FUNCTION_BLOCK "G023G_Code"
TITLE =G023G GENERAL ELEMENTS KILN MALT TRANSFER
//COPYRIGHT:    (C) 2009  BUHLER AG, CH-9240 UZWIL, SWITZERLAND
//
//PRODUCT:      WinCoS_BIW01_09
//
//TITLE:        GENERAL ELEMENTS KILN MALT TRANSFER
//                General group control
//                Allgemeine Gruppensteuerung
//
//--------------------------------------------------------------------------------
//
//IDENT:        AUTHOR:             DEPT:                              DATE:
//
//P01_FB123.1.0 K.Renz              CSB41                              29.Sep.2009
//             1st Release
//
//--------------------------------------------------------------------------------
//
//PURPOSE:
//
//MANUAL :
//
//RESTRICTIONS:
//
//--------------------------------------------------------------------------------
AUTHOR : KR
FAMILY : USW
VERSION : 9.9


VAR
  Gr : "GCS7_GrpCtrlSub";	//Standard interface to group
  InOutValue1 : DINT ;	//Data for user
  InOutValue2 : DINT ;	//Data for user
  OutWayConflict : BOOL ;	//Data for user
  OutSelectionOk : BOOL ;	//Data for user
  CmdNewValue : BOOL ;	//Data for user
  CmdNewJob : BOOL ;	//Data for user
  OutCodeOK : BOOL ;	//Data for user
  InEndOfJob : BOOL ;	//Data for user
  staWayOk : BOOL ;	//Data for user
  EdgeStartRelease : BOOL ;	//Data for user
  USW8 : BOOL ;	//Data for user
  USW9 : BOOL ;	//Data for user
  USW10 : BOOL ;	//Data for user
  USW11 : BOOL ;	//Data for user
  USW12 : BOOL ;	//Data for user
  USW13 : BOOL ;	//Data for user
  USW14 : BOOL ;	//Data for user
  USW15 : BOOL ;	//Data for user
  A_3999_SHE01 : "GCS7_E_DigInput";	// DigInpCont
  A_3999_SHE02 : "GCS7_E_DigInput";	// DigInpCont
  A_39_A040Z1 : "GCS7_E_DigInput";	// DigInpCont
  A_39_A097Z1 : "GCS7_E_DigInput";	// DigInpCont
  A_39_A187Z1 : "GCS7_E_DigInput";	// DigInpCont
  A_39_A227Z1 : "GCS7_E_DigInput";	// DigInpCont
  A_39_K091Z1 : "GCS7_E_DigInput";	// DigInpCont
  A_39_S_H097 : "GCS7_E_DigInput";	// DigInpCont
END_VAR
VAR_TEMP
  tmpEnable : BOOL ;
  tmpFlag : BOOL ;
  tmpCmdNext : BOOL ;
  tmpLocal : BOOL ;
  tmpAspOk : BOOL ;
  tmpHWStop : BOOL ;
  tmpInstanzDBNo : INT ;
END_VAR
BEGIN
NETWORK
TITLE =



NETWORK
TITLE =Read command from group control
//Parameter
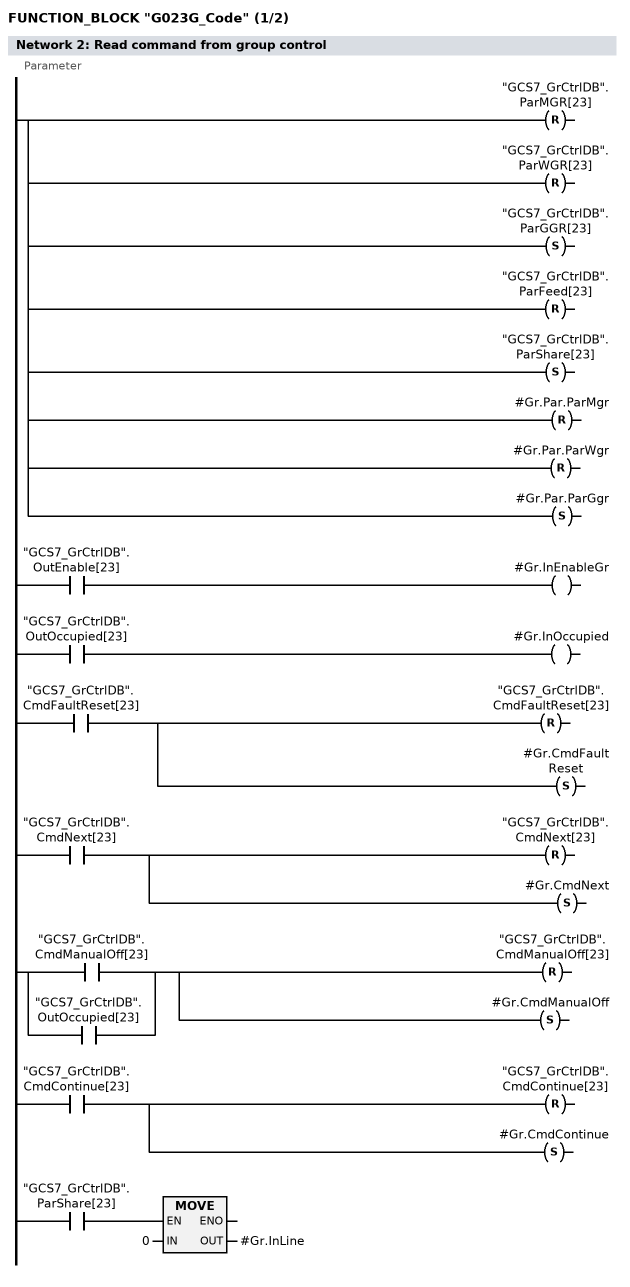
      SET   ;
      R     "GCS7_GrCtrlDB".ParMGR[23];
      R     "GCS7_GrCtrlDB".ParWGR[23];
      S     "GCS7_GrCtrlDB".ParGGR[23];
      R     "GCS7_GrCtrlDB".ParFeed[23];
      S     "GCS7_GrCtrlDB".ParShare[23];
      R     #Gr.Par.ParMgr;
      R     #Gr.Par.ParWgr;
      S     #Gr.Par.ParGgr;
//Command
      U     "GCS7_GrCtrlDB".OutEnable[23];
      =     #Gr.InEnableGr;
      U     "GCS7_GrCtrlDB".OutOccupied[23];
      =     #Gr.InOccupied;
      U     "GCS7_GrCtrlDB".CmdFaultReset[23];
      R     "GCS7_GrCtrlDB".CmdFaultReset[23];
      S     #Gr.CmdFaultReset;
      U     "GCS7_GrCtrlDB".CmdNext[23];
      R     "GCS7_GrCtrlDB".CmdNext[23];
      S     #Gr.CmdNext;
      U     "GCS7_GrCtrlDB".CmdManualOff[23];
      O     "GCS7_GrCtrlDB".OutOccupied[23];
      R     "GCS7_GrCtrlDB".CmdManualOff[23];
      S     #Gr.CmdManualOff;
      U     "GCS7_GrCtrlDB".CmdContinue[23];
      R     "GCS7_GrCtrlDB".CmdContinue[23];
      S     #Gr.CmdContinue;
//Init Line Number
      U     "GCS7_GrCtrlDB".ParShare[23];
      SPBN  WE00;
      L     0;
      T     #Gr.InLine;
WE00: NOP   0;
NETWORK
TITLE =Call Methode Control
// 1. Handle Interface PCControl
// 2. Prepare mode --> ModePassive,ModeActive,ModeIdling
// 3. Reset global flags of the group
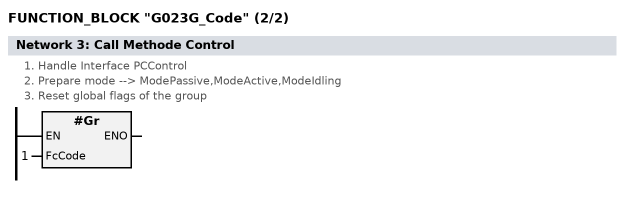
      CALL #Gr (
           FcCode                   := 1);
NETWORK
TITLE =Restart Idling Time

      CLR   ;
      S     #Gr.CmdRestartIdling;
NETWORK
TITLE =Prepare global flags



NETWORK
TITLE =Set Pattern (Target position)



NETWORK
TITLE =Interlocking WayOk



NETWORK
TITLE =Interlocking Autostart

      CLR   ;
      R     #Gr.OutAutostart;
NETWORK
TITLE =Interlocking Enable
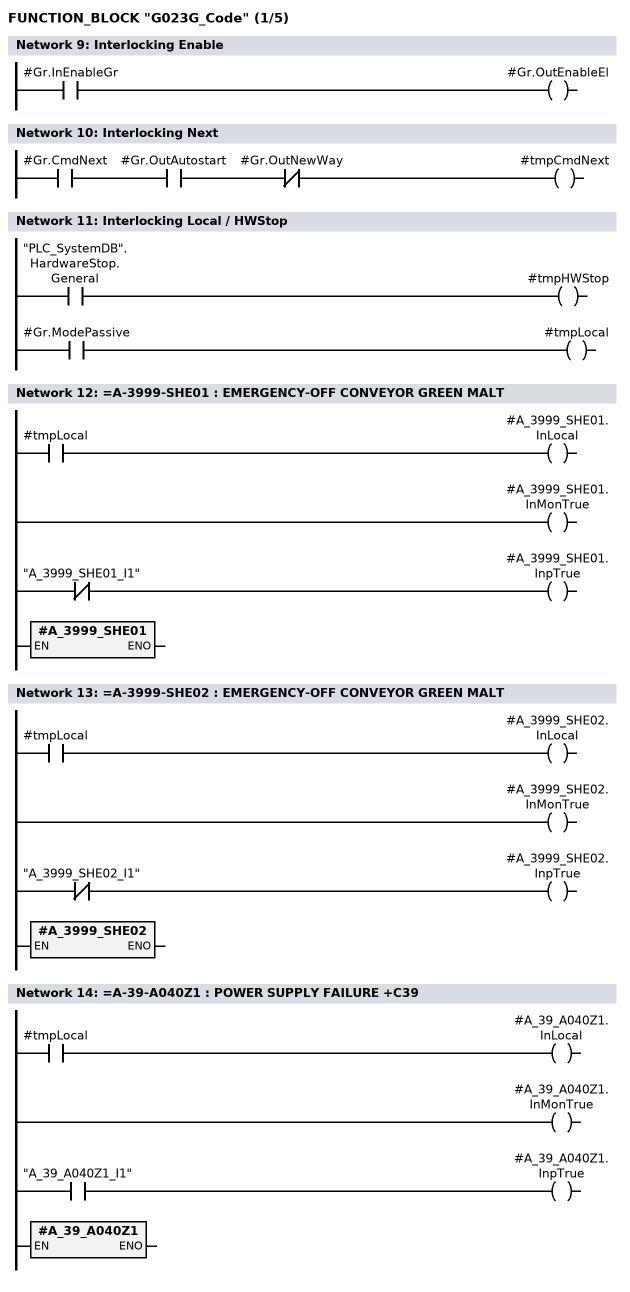

      U     #Gr.InEnableGr;
      =     #Gr.OutEnableEl;

NETWORK
TITLE =Interlocking Next

      U     #Gr.CmdNext;
      U     #Gr.OutAutostart;
      UN    #Gr.OutNewWay;
      =     #tmpCmdNext;

NETWORK
TITLE =Interlocking Local / HWStop

      U     "PLC_SystemDB".HardwareStop.General;
      =     #tmpHWStop;

      U     #Gr.ModePassive;
      =     #tmpLocal;

NETWORK
TITLE ==A-3999-SHE01 : EMERGENCY-OFF CONVEYOR GREEN MALT

      NOP   0;
//-InLocal---
      U     #tmpLocal;
      =     #A_3999_SHE01.InLocal;
//
//-Monitoring---
      SET   ;
      =     #A_3999_SHE01.InMonTrue;
//
//-PreAlarm---
//  CLR
//  =      #A_3999_SHE01.InPreAlarmTrue
//
//-Additional commands---
//      CLR
//      S     #A_3999_SHE01.CmdRunTimeOutTime
//
//-Read inputs---
      UN    "A_3999_SHE01_I1";
      =     #A_3999_SHE01.InpTrue;
//
//-Set Parameters---
//
//-Call object control---
      CALL #A_3999_SHE01 ;
//
//-Write outputs---
NETWORK
TITLE ==A-3999-SHE02 : EMERGENCY-OFF CONVEYOR GREEN MALT

      NOP   0;
//-InLocal---
      U     #tmpLocal;
      =     #A_3999_SHE02.InLocal;
//
//-Monitoring---
      SET   ;
      =     #A_3999_SHE02.InMonTrue;
//
//-PreAlarm---
//  CLR
//  =      #A_3999_SHE02.InPreAlarmTrue
//
//-Additional commands---
//      CLR
//      S     #A_3999_SHE02.CmdRunTimeOutTime
//
//-Read inputs---
      UN    "A_3999_SHE02_I1";
      =     #A_3999_SHE02.InpTrue;
//
//-Set Parameters---
//
//-Call object control---
      CALL #A_3999_SHE02 ;
//
//-Write outputs---
NETWORK
TITLE ==A-39-A040Z1 : POWER SUPPLY FAILURE +C39

      NOP   0;
//-InLocal---
      U     #tmpLocal;
      =     #A_39_A040Z1.InLocal;
//
//-Monitoring---
      SET   ;
      =     #A_39_A040Z1.InMonTrue;
//
//-PreAlarm---
//  CLR
//  =      #A_39_A040Z1.InPreAlarmTrue
//
//-Additional commands---
//      CLR
//      S     #A_39_A040Z1.CmdRunTimeOutTime
//
//-Read inputs---
      U     "A_39_A040Z1_I1";
      =     #A_39_A040Z1.InpTrue;
//
//-Set Parameters---
//
//-Call object control---
      CALL #A_39_A040Z1 ;
//
//-Write outputs---
NETWORK
TITLE ==A-39-A097Z1 : EMERGENCY-STOP +C39
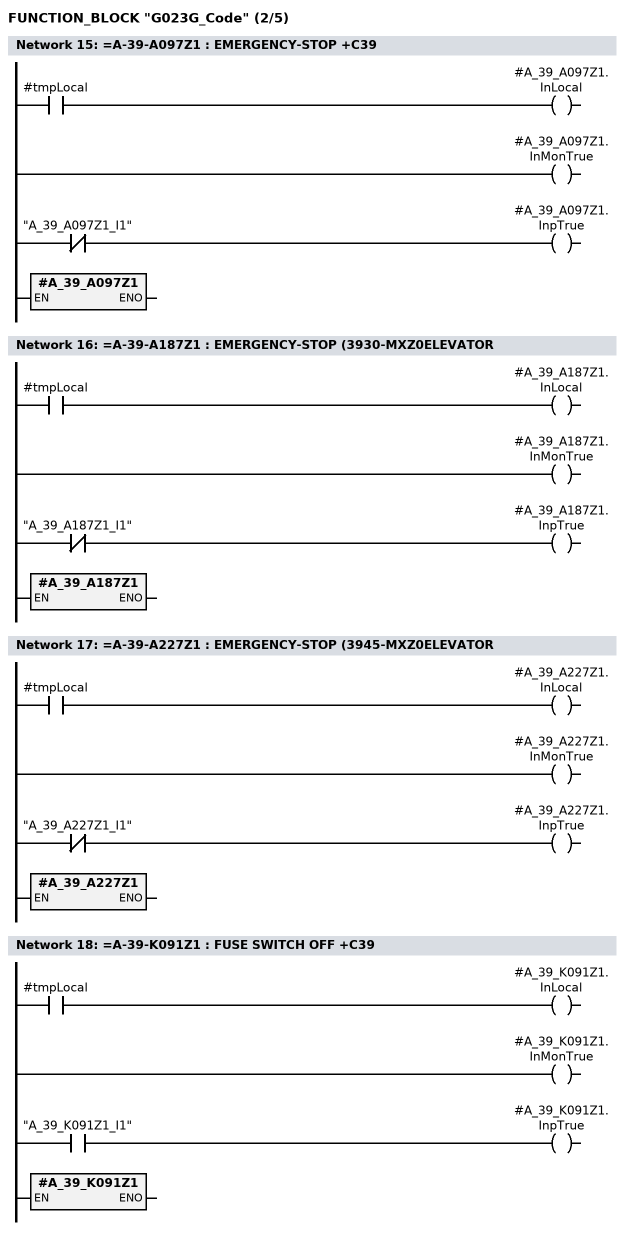

      NOP   0;
//-InLocal---
      U     #tmpLocal;
      =     #A_39_A097Z1.InLocal;
//
//-Monitoring---
      SET   ;
      =     #A_39_A097Z1.InMonTrue;
//
//-PreAlarm---
//  CLR
//  =      #A_39_A097Z1.InPreAlarmTrue
//
//-Additional commands---
//      CLR
//      S     #A_39_A097Z1.CmdRunTimeOutTime
//
//-Read inputs---
//MW 2010.04.16      U     "A_39_A097Z1_I1"
      UN    "A_39_A097Z1_I1";
      =     #A_39_A097Z1.InpTrue;
//
//-Set Parameters---
//
//-Call object control---
      CALL #A_39_A097Z1 ;
//
//-Write outputs---
NETWORK
TITLE ==A-39-A187Z1 : EMERGENCY-STOP (3930-MXZ0ELEVATOR

      NOP   0;
//-InLocal---
      U     #tmpLocal;
      =     #A_39_A187Z1.InLocal;
//
//-Monitoring---
      SET   ;
      =     #A_39_A187Z1.InMonTrue;
//
//-PreAlarm---
//  CLR
//  =      #A_39_A187Z1.InPreAlarmTrue
//
//-Additional commands---
//      CLR
//      S     #A_39_A187Z1.CmdRunTimeOutTime
//
//-Read inputs---
      UN    "A_39_A187Z1_I1";
      =     #A_39_A187Z1.InpTrue;
//
//-Set Parameters---
//
//-Call object control---
      CALL #A_39_A187Z1 ;
//
//-Write outputs---
NETWORK
TITLE ==A-39-A227Z1 : EMERGENCY-STOP (3945-MXZ0ELEVATOR

      NOP   0;
//-InLocal---
      U     #tmpLocal;
      =     #A_39_A227Z1.InLocal;
//
//-Monitoring---
      SET   ;
      =     #A_39_A227Z1.InMonTrue;
//
//-PreAlarm---
//  CLR
//  =      #A_39_A227Z1.InPreAlarmTrue
//
//-Additional commands---
//      CLR
//      S     #A_39_A227Z1.CmdRunTimeOutTime
//
//-Read inputs---
      UN    "A_39_A227Z1_I1";
      =     #A_39_A227Z1.InpTrue;
//
//-Set Parameters---
//
//-Call object control---
      CALL #A_39_A227Z1 ;
//
//-Write outputs---
NETWORK
TITLE ==A-39-K091Z1 : FUSE SWITCH OFF +C39

      NOP   0;
//-InLocal---
      U     #tmpLocal;
      =     #A_39_K091Z1.InLocal;
//
//-Monitoring---
      SET   ;
      =     #A_39_K091Z1.InMonTrue;
//
//-PreAlarm---
//  CLR
//  =      #A_39_K091Z1.InPreAlarmTrue
//
//-Additional commands---
//      CLR
//      S     #A_39_K091Z1.CmdRunTimeOutTime
//
//-Read inputs---
      U     "A_39_K091Z1_I1";
      =     #A_39_K091Z1.InpTrue;
//
//-Set Parameters---
//
//-Call object control---
      CALL #A_39_K091Z1 ;
//
//-Write outputs---
NETWORK
TITLE ==A-39-S/H097 : OPERATING ON +C39
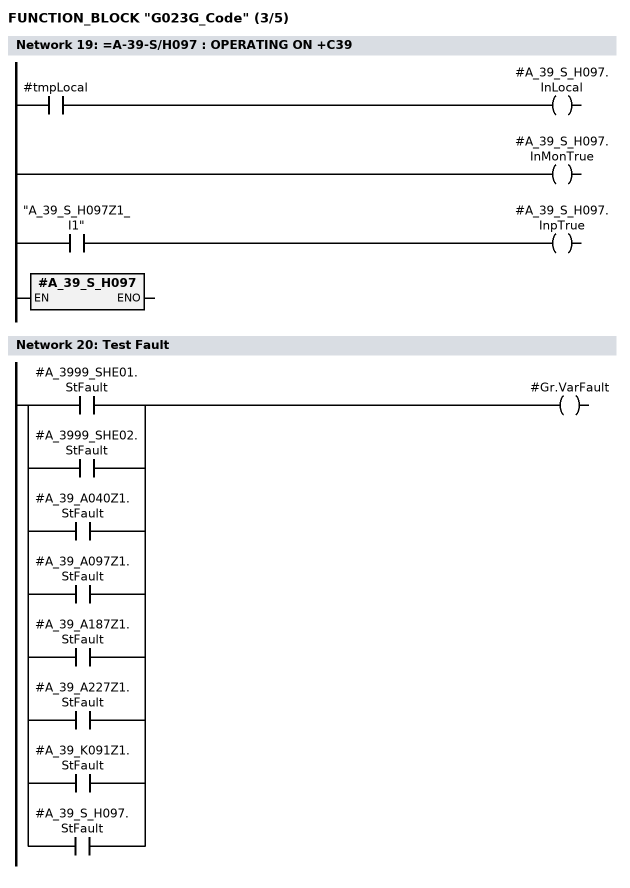

      NOP   0;
//-InLocal---
      U     #tmpLocal;
      =     #A_39_S_H097.InLocal;
//
//-Monitoring---
      SET   ;
      =     #A_39_S_H097.InMonTrue;
//
//-PreAlarm---
//  CLR
//  =      #A_39_S_H097.InPreAlarmTrue
//
//-Additional commands---
//      CLR
//      S     #A_39_S_H097.CmdRunTimeOutTime
//
//-Read inputs---
      U     "A_39_S_H097Z1_I1";
      =     #A_39_S_H097.InpTrue;
//
//-Set Parameters---
//
//-Call object control---
      CALL #A_39_S_H097 ;
//
//-Write outputs---
NETWORK
TITLE =Test Fault

      U     #A_3999_SHE01.StFault;
      O     #A_3999_SHE02.StFault;
      O     #A_39_A040Z1.StFault;
      O     #A_39_A097Z1.StFault;
      O     #A_39_A187Z1.StFault;
      O     #A_39_A227Z1.StFault;
      O     #A_39_K091Z1.StFault;
      O     #A_39_S_H097.StFault;
      =     #Gr.VarFault;
NETWORK
TITLE =Test Warning
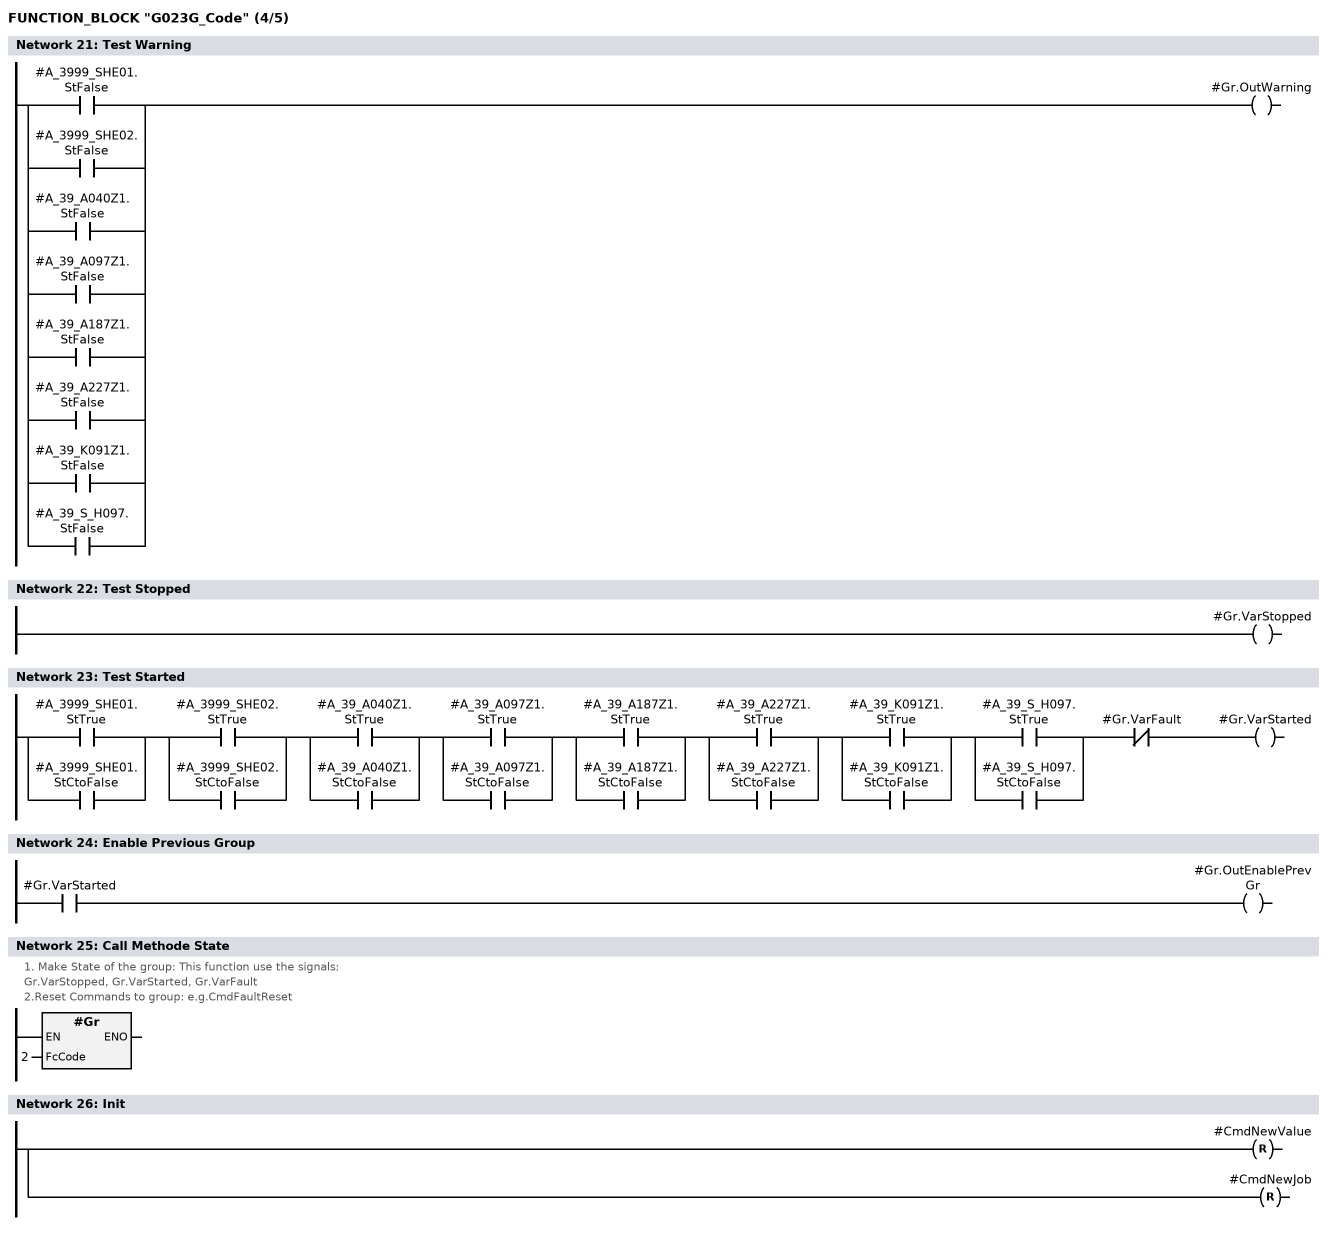

      U     #A_3999_SHE01.StFalse;
      O     #A_3999_SHE02.StFalse;
      O     #A_39_A040Z1.StFalse;
      O     #A_39_A097Z1.StFalse;
      O     #A_39_A187Z1.StFalse;
      O     #A_39_A227Z1.StFalse;
      O     #A_39_K091Z1.StFalse;
      O     #A_39_S_H097.StFalse;
      =     #Gr.OutWarning;
NETWORK
TITLE =Test Stopped

      SET   ;
      =     #Gr.VarStopped;
NETWORK
TITLE =Test Started

      U(    ;
      O     #A_3999_SHE01.StTrue;
      O     #A_3999_SHE01.StCtoFalse;
      )     ;
      U(    ;
      O     #A_3999_SHE02.StTrue;
      O     #A_3999_SHE02.StCtoFalse;
      )     ;
      U(    ;
      O     #A_39_A040Z1.StTrue;
      O     #A_39_A040Z1.StCtoFalse;
      )     ;
      U(    ;
      O     #A_39_A097Z1.StTrue;
      O     #A_39_A097Z1.StCtoFalse;
      )     ;
      U(    ;
      O     #A_39_A187Z1.StTrue;
      O     #A_39_A187Z1.StCtoFalse;
      )     ;
      U(    ;
      O     #A_39_A227Z1.StTrue;
      O     #A_39_A227Z1.StCtoFalse;
      )     ;
      U(    ;
      O     #A_39_K091Z1.StTrue;
      O     #A_39_K091Z1.StCtoFalse;
      )     ;
      U(    ;
      O     #A_39_S_H097.StTrue;
      O     #A_39_S_H097.StCtoFalse;
      )     ;
      UN    #Gr.VarFault;
      =     #Gr.VarStarted;
NETWORK
TITLE =Enable Previous Group

      U     #Gr.VarStarted;
      =     #Gr.OutEnablePrevGr;
NETWORK
TITLE =Call Methode State
//1. Make State of the group: This function use the signals:
//        Gr.VarStopped, Gr.VarStarted, Gr.VarFault
//2.Reset Commands to group: e.g.CmdFaultReset
      CALL #Gr (
           FcCode                   := 2);
NETWORK
TITLE =Init

      SET   ;
      R     #CmdNewValue;
      R     #CmdNewJob;
NETWORK
TITLE =Write data to group control
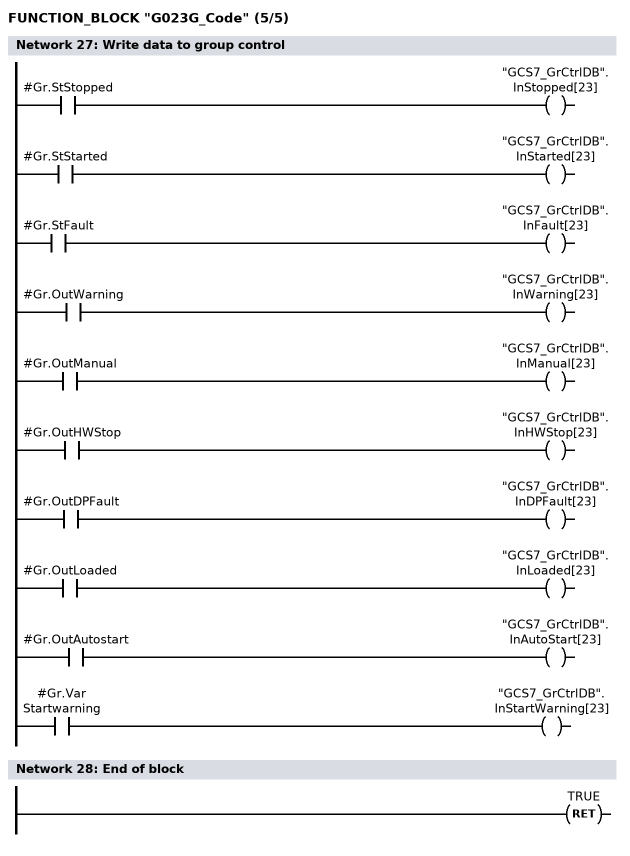

      U     #Gr.StStopped;
      =     "GCS7_GrCtrlDB".InStopped[23];
      U     #Gr.StStarted;
      =     "GCS7_GrCtrlDB".InStarted[23];
      U     #Gr.StFault;
      =     "GCS7_GrCtrlDB".InFault[23];
      U     #Gr.OutWarning;
      =     "GCS7_GrCtrlDB".InWarning[23];
      U     #Gr.OutManual;
      =     "GCS7_GrCtrlDB".InManual[23];
      U     #Gr.OutHWStop;
      =     "GCS7_GrCtrlDB".InHWStop[23];
      U     #Gr.OutDPFault;
      =     "GCS7_GrCtrlDB".InDPFault[23];
      U     #Gr.OutLoaded;
      =     "GCS7_GrCtrlDB".InLoaded[23];
      U     #Gr.OutAutostart;
      =     "GCS7_GrCtrlDB".InAutoStart[23];
      U     #Gr.VarStartwarning;
      =     "GCS7_GrCtrlDB".InStartWarning[23];
NETWORK
TITLE =End of block

      BE    ;

END_FUNCTION_BLOCK

